FUNCTION_BLOCK FB_FANUC_Basic
VAR_INPUT
END_VAR
VAR_OUTPUT
	qEnable:BOOL;
	qFault:BOOL;
END_VAR
VAR
	_rawIn AT %I*:ARRAY[0..7]OF BYTE;
	_rawOut AT %Q*:ARRAY[0..7]OF BYTE;
	_EIPConnectionState AT %i*:UINT;
	_UI1:DUT_FANUC_UI1;
	_UO1:DUT_FANUC_UO1;
END_VAR

METHOD PUBLIC Enable : BOOL
VAR_INPUT
	iTrigger:BOOL;
END_VAR
VAR
	_RobotEnable:BOOL;
END_VAR
_RobotEnable:=iTrigger AND NOT Fault();

_UI1.UI01_IMSP:=_RobotEnable;
_UI1.UI03_SFSP:=_RobotEnable;
_UI1.UI08_Enable:=_RobotEnable;
_UI1.UI02_Hold:=_RobotEnable;
END_METHOD

METHOD PROTECTED Fault : BOOL
VAR_INPUT
END_VAR
Fault:=_UO1.UO06_Fault OR _UO1.UO09_BattAlarm;
END_METHOD

METHOD PUBLIC Reset : BOOL
VAR_INPUT
	iTrigger:BOOL;
END_VAR
_UI1.UI05_FaultReset:=iTrigger;
END_METHOD

METHOD PUBLIC Update : BOOL
MEMMOVE(
destAddr:=ADR(_UO1)
,srcAddr:=ADR(_rawIn[0])
,n:=4
);


MEMMOVE(
destAddr:=ADR(_rawOut[0])
,srcAddr:=ADR(_UI1)
,n:=4
);


qEnable:=_UO1.UO01_CmdEnabled AND _UO1.UO02_SystemReady;
qFault:=Fault();
END_METHOD

END_FUNCTION_BLOCK

(* stored: Version 1.1.0.1, ProductVersion 3.1.4024.15
   POU FB_FANUC_Basic: Id {d8361be0-a695-4cd7-af64-af0d44a691af}, SpecialFunc None
   Method Enable: Id {0bf52179-a93a-4419-870a-1b3de78b9461}
   Method Fault: Id {4b1010de-e02c-43d3-b09d-7bc403f827ff}
   Method Reset: Id {4f2083e8-6a7e-44e8-b73b-821d2cdaeea0}
   Method Update: Id {958b983e-3529-4d9f-90a3-b98c26734e48} *)
